Yaskawa INFORM job: TCP_R1.JBI

/JOB
//NAME TCP_R1
///FOLDERNAME SAFETY
//POS
///NPOS 6,6,0,0,0,0
///TOOL 0
///POSTYPE PULSE
///PULSE
C00000=25422,122237,13311,-12237,93772,84182
C00001=22558,137824,39586,-10513,85519,84319
C00002=22559,138155,40658,-10516,85040,84359
C00003=20973,136718,38421,-9578,85532,83947
C00004=20973,138060,39146,-9576,85772,83929
C00005=25422,122237,13311,-12237,93772,84182
BC00000=125179,23837,1075001
BC00001=147637,23837,1075001
BC00002=147637,23837,1075001
BC00003=147637,23837,1075001
BC00004=147637,23837,1075001
BC00005=125179,23837,1075001
//INST
///DATE 2023/12/06 11:05
///ATTR SC,RW
///GROUP1 RB1,BS1
NOP
MOVJ C00000 BC00000 VJ=10.00
MOVJ C00001 BC00001 VJ=10.00
MOVL C00002 BC00002 V=11.0
MOVL C00003 BC00003 V=11.0
PAUSE
MOVJ C00004 BC00004 VJ=10.00
MOVJ C00005 BC00005 VJ=10.00
END
